FUNCTION_BLOCK FB_ApplyLocks
VAR_INPUT
	isStationLocked:BOOL;
END_VAR
VAR_OUTPUT
END_VAR
VAR
END_VAR
VAR_IN_OUT
		stationState:typeStationMode;
END_VAR

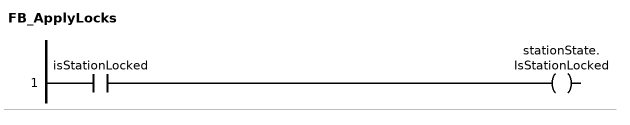
// NETWORK 1
stationState.IsStationLocked := isStationLocked;

END_FUNCTION_BLOCK

(* stored: Version 1.1.0.1, ProductVersion 3.1.4024.11
   POU FB_ApplyLocks: Id {2678a292-78e2-0d13-3502-ad8dd52710e8}, SpecialFunc None *)
